// TIA Portal V17 export
// export: Created 2025-03-05T08:02:22.859126Z, ExportSetting WithDefaults, DisplayName Totally Integrated Automation Portal, DisplayVersion V17 Update 8, DisplayName TIA Portal Openness, DisplayVersion V17 Update 8, DisplayName TIA Portal Version Control Interface, DisplayVersion V17, DisplayName SINAMICS Startdrive Advanced, DisplayVersion V17 SP2, DisplayName SINAMICS Startdrive G110M, G120, G120C, G120D, G120P, G115D, DisplayVersion V17 SP2, DisplayName SINAMICS Startdrive G130, G150, S120, S150, SINAMICS MV, S210, DisplayVersion V17 SP2, DisplayName STEP 7 Professional, DisplayVersion V17 Update 8, DisplayName SINUMERIK ONE STEP 7 Toolbox, DisplayVersion V17 Update 12, DisplayName SINUMERIK 840D sl STEP 7 Toolbox, DisplayVersion V17 Update 12, DisplayName STEP 7 Safety, DisplayVersion V17 Update 6, DisplayName WinCC Advanced, DisplayVersion V17 Update 8
TYPE "CHANNEL_PLC_SIGNALS"
// stored: IsFailsafeCompliant false
   STRUCT
      INPUT : Struct
         START_POSITION_SIGNAL : Bool;
         RETURN_HOME_SIGNAL : Bool;
         START_TORQUE_SIGNAL : Bool;
      END_STRUCT;
      OUTPUT : Struct
         IN_POSITION_SIGNAL : Bool;
         IN_HOME_SIGNAL : Bool;
         IN_TORQUE_SIGNAL : Bool;
      END_STRUCT;
   END_STRUCT;
END_TYPE
